(* PLC project ST_FOR_AND_CASE_2, Beckhoff Automation GmbH TwinCAT PLC Control 3.5.10.30 *)
(* stored: creationDateTime 2019-09-26T11:42:34.782397, modificationDateTime 2019-09-26T11:42:34.7853953 *)

PROGRAM MAIN
VAR

	Present: INT;
	Open: INT;
	Close: INT;
	Workpiece: BOOL;
	SENSOR: BOOL;
	Gate: INT;
END_VAR

                  

FOR counter:= 2 TO 5 BY 1 DO
	CASE counter OF
	1, 3:  
		BOOL1 := TRUE;
	2:     
		BOOL2 := FALSE;
	ELSE
		BOOL1 := NOT BOOL1;
	END_CASE;
END_FOR;


                
END_PROGRAM

CONFIGURATION Application
  RESOURCE ST_Evolution_1 ON PLC
    TASK PlcTask(INTERVAL := T#0ms, PRIORITY := 20);
    PROGRAM MAIN WITH PlcTask : MAIN;
  END_RESOURCE
END_CONFIGURATION
